FUNCTION_BLOCK FB_SafeInfoState
VAR
	State AT%I* :USINT;
	Diag AT%I* :UINT;
END_VAR

END_FUNCTION_BLOCK

(* stored: Version 1.1.0.1, ProductVersion 3.1.4024.12
   POU FB_SafeInfoState: Id {7b354806-906f-4406-9f13-596985335ebb}, SpecialFunc None *)
